TYPE
    RackStatus : STRUCT
        available : BOOL;
        blocked   : BOOL;
    END_STRUCT
END_TYPE

(* stored: Version 1.1.0.1
   DUT RackStatus: Id {d80071a5-2851-4e8a-81a5-a71433ab7f21} *)
